INTERFACE I_AxisDynamics EXTENDS __SYSTEM.IQueryInterface

PROPERTY PUBLIC Acceleration : mc_lreal
GET
END_GET
SET
END_SET
END_PROPERTY

PROPERTY BufferMode : MC_BufferMode
GET
END_GET
SET
END_SET
END_PROPERTY

PROPERTY PUBLIC Deceleration : mc_lreal
GET
END_GET
SET
END_SET
END_PROPERTY

PROPERTY PUBLIC Jerk : mc_lreal
GET
END_GET
SET
END_SET
END_PROPERTY

END_INTERFACE

(* stored: Version 1.1.0.1
   Itf I_AxisDynamics: Id {f3908ec5-f9cc-47a8-9ad5-05c8b414800b}
   Property Acceleration: Id {72d27c44-987d-44ce-a99c-48cb32673553}
   Get Get: Id {056425fd-3278-4643-be11-9a6970fe13ef}
   Set Set: Id {9650a87b-bd43-4b24-b18c-102d81cc67c2}
   Property BufferMode: Id {ced436f6-287e-418d-af69-e4b848d62760}
   Get Get: Id {0f0cbae8-b515-46ff-8f32-af99ff57dd92}
   Set Set: Id {17cb71bf-508b-4dc2-9600-83c2f4af678e}
   Property Deceleration: Id {5ef3957c-6644-426d-8ede-03dbef11af09}
   Get Get: Id {bffc68c4-d0c8-4caa-bb08-1acb04f5a311}
   Set Set: Id {615e48f2-1833-4891-bf53-66cbe72eae8a}
   Property Jerk: Id {dd32e94c-e653-4f44-ba1a-16a122c64a8f}
   Get Get: Id {ed85520a-8680-4906-88bb-bb44509a959d}
   Set Set: Id {4339837f-910b-4c9c-913e-e3f9f3195613} *)
